FUNCTION Convert_BOOL_TO_LREAL : Hresult
VAR_INPUT
	in : BOOL;
	out : REFERENCE TO LREAL;
END_VAR
VAR
	converted : LREAL;
END_VAR

converted := BOOL_TO_LREAL(in);

IF (LREAL_TO_BOOL(converted) <> in) THEN
	Convert_BOOL_TO_LREAL := INCOMPATIBLE;
	RETURN;
END_IF

out := converted;

END_FUNCTION

(* stored: Version 1.1.0.1, ProductVersion 3.1.4024.12
   POU Convert_BOOL_TO_LREAL: Id {3e8fe6b6-59db-4930-baf1-543fc94bd8fc}, SpecialFunc None *)
